FUNCTION_BLOCK CTU_OUT (* E_CTU with display and label *)
  (* Standard: 61499-2 *)
  (* Version 0.0, 2004-08-07, JHC, Rockwell Automation *)
  (* Compiler header: package fb.rt.swing; *)
  (* Compiler Java Sun JDK 1.4.2 *)
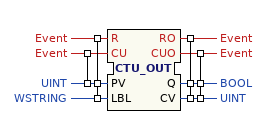
  EVENT_INPUT
    R WITH PV, LBL; (* Reset Counter and Initialize Display *)
    CU WITH PV; (* Count Up *)
  END_EVENT
  EVENT_OUTPUT
    RO WITH CV, Q; (* Counter Reset *)
    CUO WITH CV, Q; (* Count Up Output Event *)
  END_EVENT
  VAR_INPUT
    PV : UINT; (* Preset Value *)
    LBL : WSTRING; (* Label *)
  END_VAR
  VAR_OUTPUT
    Q : BOOL; (* CV>=PV *)
    CV : UINT; (* Counter Value *)
  END_VAR
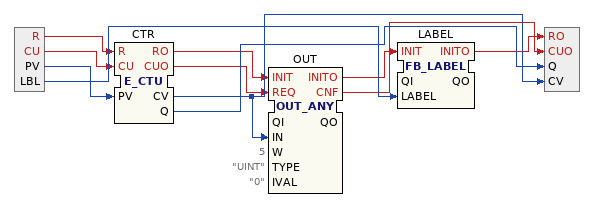
  FBS
    CTR : E_CTU;
    OUT : OUT_ANY(IVAL := "0", TYPE := "UINT", W := 5);
    LABEL : FB_LABEL;
  END_FBS
  EVENT_CONNECTIONS
    CTR.RO TO OUT.INIT;
    CTR.CUO TO OUT.REQ;
    R TO CTR.R;
    CU TO CTR.CU;
    OUT.CNF TO CUO;
    OUT.INITO TO LABEL.INIT;
    LABEL.INITO TO RO;
  END_CONNECTIONS
  DATA_CONNECTIONS
    CTR.CV TO OUT.IN;
    CTR.CV TO CV;
    PV TO CTR.PV;
    CTR.Q TO Q;
    LBL TO LABEL.LABEL;
  END_CONNECTIONS
END_FUNCTION_BLOCK
